PROGRAM PRG_GEM1_42
VAR
	
	
END_VAR

END_PROGRAM

(* stored: Version 1.1.0.1, ProductVersion 3.1.4022.16
   POU PRG_GEM1_42: Id {93631957-4630-41b1-9ec4-9b9aeaf56294}, SpecialFunc None *)
